FUNCTION_BLOCK FB_FCSLComponentBase EXTENDS FB_ComponentBase

VAR

END_VAR

METHOD M_AuditLog : HRESULT

VAR_INPUT
	k : T_MaxString;
	v : T_MaxString;
END_VAR
GVL_FCSLTracing.auditLog.M_AddEntry(k := k, v := v);

M_AuditLog := S_OK;
END_METHOD

METHOD M_SysLog : HRESULT

VAR_INPUT
	msg 			: T_MaxString;
	debug 			: E_SysLogLevel;
END_VAR

VAR
	debugString 	: STRING;
	debugINT 		: UDINT;
	json 			: T_MaxString;	
END_VAR
IF ( debug = E_SysLogLevel.invalid ) THEN
	RETURN;
END_IF

// Send log entry
GVL_FCSLTracing.sysLog.M_AddEntry(
    Source := InstancePath, 
    Message := msg, 
    logLevel := debug, 
    Flags := 0
);

// Return success
M_SysLog := S_OK;
END_METHOD

END_FUNCTION_BLOCK

(* stored: Version 1.1.0.1
   POU FB_FCSLComponentBase: Id {293810a7-d588-4a02-bf97-9f4610062714}, SpecialFunc None
   Method M_AuditLog: Id {abb9e373-22da-47da-a2c3-e3f1e7cd875a}
   Method M_SysLog: Id {b4fab106-d19e-44ac-9789-66501b183208} *)
